// TIA Portal V16 export
// export: Created 2021-09-01T13:50:45.6587865Z, ExportSetting WithDefaults, DisplayName Totally Integrated Automation Portal, DisplayVersion V16 Update 3, DisplayName TIA Portal Version Control Interface, DisplayVersion V16 Update 2, DisplayName TIA Portal Openness, DisplayVersion V16 Update 3, DisplayName TIA Portal Teamcenter Gateway, DisplayVersion V16, DisplayName STEP 7 Professional, DisplayVersion V16 Update 3, DisplayName STEP 7 Safety, DisplayVersion V16, DisplayName WinCC Advanced, DisplayVersion V16 Update 3
TYPE "UF_FLAGS"
// stored: IsFailsafeCompliant false
   STRUCT
      NotAvaible : Bool;
      Stop : Bool;
      Work : Bool;
      HW : Bool;
      HWa : Bool;
      CEB1 : Bool;
      CEB1a : Bool;
      CEB2 : Bool;
      CEB2a : Bool;
      Soak : Bool;
      Err : Bool;
      ErrWork : Bool;
      ErrHW : Bool;
      ErrCEB1 : Bool;
      ErrCEB2 : Bool;
      Spare_1 : Bool;
   END_STRUCT;
END_TYPE
